// TIA Portal V16 export
// export: Created 2024-12-03T15:41:39.243873Z, ExportSetting WithDefaults, DisplayName Totally Integrated Automation Portal, DisplayVersion V16 Update 6, DisplayName TIA Portal Version Control Interface, DisplayVersion V16 Update 2, DisplayName TIA Portal Openness, DisplayVersion V16 Update 6, DisplayName TIA Portal Teamcenter Gateway, DisplayVersion V16, DisplayName SINAMICS Startdrive Advanced, DisplayVersion V16 Update 5, DisplayName SINAMICS Startdrive G130, G150, S120, S150, SINAMICS MV, S210, DisplayVersion V16 Update 5, DisplayName SINAMICS Startdrive G110M, G120, G120C, G120D, G120P, G115D, DisplayVersion V16 Update 5, DisplayName STEP 7 Professional, DisplayVersion V16 Update 6, DisplayName STEP 7 Safety, DisplayVersion V16, DisplayName WinCC Advanced / Unified PC, DisplayVersion V16 Update 6
FUNCTION_BLOCK "InputReaderConveyLinx_FB"   // FB127, SCL
{ S7_Optimized_Access := 'TRUE' }
VERSION : 0.1
// stored: AutoNumber true, IsIECCheckEnabled false, IsRetainMemResEnabled false, MemoryReserve 100, SetENOAutomatically false, UDAEnableTagReadback false
   VAR
      FTC_102_L2 : "SmartBool";
      FTC_102_L4 : "SmartBool";
      FTC_102_R2 : "SmartBool";
      FTC_102_R4 : "SmartBool";
      FTC_103_L2 : "SmartBool";
      FTC_103_L4 : "SmartBool";
      FTC_103_R2 : "SmartBool";
      FTC_103_R4 : "SmartBool";
      FTC_104_L2 : "SmartBool";
      FTC_104_L4 : "SmartBool";
      FTC_104_R2 : "SmartBool";
      FTC_104_R4 : "SmartBool";
      FTC_105_L2 : "SmartBool";
      FTC_105_L4 : "SmartBool";
      FTC_105_R2 : "SmartBool";
      FTC_105_R4 : "SmartBool";
      FTC_106_L2 : "SmartBool";
      FTC_106_L4 : "SmartBool";
      FTC_106_R2 : "SmartBool";
      FTC_106_R4 : "SmartBool";
      FTC_107_L2 : "SmartBool";
      FTC_107_L4 : "SmartBool";
      FTC_107_R2 : "SmartBool";
      FTC_107_R4 : "SmartBool";
      FTC_108_L2 : "SmartBool";
      FTC_108_L4 : "SmartBool";
      FTC_108_R2 : "SmartBool";
      FTC_108_R4 : "SmartBool";
      FTC_109_L2 : "SmartBool";
      FTC_109_L4 : "SmartBool";
      FTC_109_R2 : "SmartBool";
      FTC_109_R4 : "SmartBool";
      FTC_110_L2 : "SmartBool";
      FTC_110_L4 : "SmartBool";
      FTC_110_R2 : "SmartBool";
      FTC_110_R4 : "SmartBool";
      FTC_111_L2 : "SmartBool";
      FTC_111_L4 : "SmartBool";
      FTC_111_R2 : "SmartBool";
      FTC_111_R4 : "SmartBool";
      FTC_112_L2 : "SmartBool";
      FTC_112_L4 : "SmartBool";
      FTC_112_R2 : "SmartBool";
      FTC_112_R4 : "SmartBool";
      FTC_113_L2 : "SmartBool";
      FTC_113_L4 : "SmartBool";
      FTC_113_R2 : "SmartBool";
      FTC_113_R4 : "SmartBool";
      FTC_114_L2 : "SmartBool";
      FTC_114_L4 : "SmartBool";
      FTC_114_R2 : "SmartBool";
      FTC_114_R4 : "SmartBool";
      FTC_115_L2 : "SmartBool";
      FTC_115_L4 : "SmartBool";
      FTC_115_R2 : "SmartBool";
      FTC_115_R4 : "SmartBool";
      FTC_202_L2 : "SmartBool";
      FTC_202_L4 : "SmartBool";
      FTC_202_R2 : "SmartBool";
      FTC_202_R4 : "SmartBool";
      FTC_203_L2 : "SmartBool";
      FTC_203_L4 : "SmartBool";
      FTC_203_R2 : "SmartBool";
      FTC_203_R4 : "SmartBool";
      FTC_301_L2 : "SmartBool";
      FTC_301_L4 : "SmartBool";
      FTC_301_R2 : "SmartBool";
      FTC_301_R4 : "SmartBool";
      FTC_302_L2 : "SmartBool";
      FTC_302_L4 : "SmartBool";
      FTC_302_R2 : "SmartBool";
      FTC_302_R4 : "SmartBool";
      FTC_303_L2 : "SmartBool";
      FTC_303_L4 : "SmartBool";
      FTC_303_R2 : "SmartBool";
      FTC_303_R4 : "SmartBool";
      FTC_304_L2 : "SmartBool";
      FTC_304_L4 : "SmartBool";
      FTC_304_R2 : "SmartBool";
      FTC_304_R4 : "SmartBool";
      FTC_305_L2 : "SmartBool";
      FTC_305_L4 : "SmartBool";
      FTC_305_R2 : "SmartBool";
      FTC_305_R4 : "SmartBool";
   END_VAR
BEGIN
   REGION CON_102 

       #FTC_102_L2(I_Sensor := NOT "I_CON_102".AllSensors.LeftPin2,
                   O_data => "Inputs_DB".FTC_102_L2);

       #FTC_102_L4(I_Sensor := NOT "I_CON_102".AllSensors.LeftPin4,
                   O_data => "Inputs_DB".FTC_102_L4);

       #FTC_102_R2(I_Sensor := NOT "I_CON_102".AllSensors.RightPin2,
                   O_data => "Inputs_DB".FTC_102_R2);

       #FTC_102_R4(I_Sensor := NOT "I_CON_102".AllSensors.RightPin4,
                   O_data => "Inputs_DB".FTC_102_R4);

   END_REGION

   REGION CON_103 

       #FTC_103_L2(I_Sensor := NOT "I_CON_103".AllSensors.LeftPin2,
                   O_data => "Inputs_DB".FTC_103_L2);

       #FTC_103_L4(I_Sensor := NOT "I_CON_103".AllSensors.LeftPin4,
                   O_data => "Inputs_DB".FTC_103_L4);

       #FTC_103_R2(I_Sensor := NOT "I_CON_103".AllSensors.RightPin2,
                   O_data => "Inputs_DB".FTC_103_R2);

       #FTC_103_R4(I_Sensor := NOT "I_CON_103".AllSensors.RightPin4,
                   O_data => "Inputs_DB".FTC_103_R4);

   END_REGION

   REGION CON_104 

       #FTC_104_L2(I_Sensor := NOT "I_CON_104".AllSensors.LeftPin2,
                   O_data => "Inputs_DB".FTC_104_L2);

       #FTC_104_L4(I_Sensor := NOT "I_CON_104".AllSensors.LeftPin4,
                   O_data => "Inputs_DB".FTC_104_L4);

       #FTC_104_R2(I_Sensor := NOT "I_CON_104".AllSensors.RightPin2,
                   O_data => "Inputs_DB".FTC_104_R2);

       #FTC_104_R4(I_Sensor := NOT "I_CON_104".AllSensors.RightPin4,
                   O_data => "Inputs_DB".FTC_104_R4);

   END_REGION

   REGION CON_105 

       #FTC_105_L2(I_Sensor := NOT "I_CON_105".AllSensors.LeftPin2,
                   O_data => "Inputs_DB".FTC_105_L2);

       #FTC_105_L4(I_Sensor := NOT "I_CON_105".AllSensors.LeftPin4,
                   O_data => "Inputs_DB".FTC_105_L4);

       #FTC_105_R2(I_Sensor := NOT "I_CON_105".AllSensors.RightPin2,
                   O_data => "Inputs_DB".FTC_105_R2);

       #FTC_105_R4(I_Sensor := NOT "I_CON_105".AllSensors.RightPin4,
                   O_data => "Inputs_DB".FTC_105_R4);

   END_REGION

   REGION CON_106 

       #FTC_106_L2(I_Sensor := NOT "I_CON_106".AllSensors.LeftPin2,
                   O_data => "Inputs_DB".FTC_106_L2);

       #FTC_106_L4(I_Sensor := NOT "I_CON_106".AllSensors.LeftPin4,
                   O_data => "Inputs_DB".FTC_106_L4);

       #FTC_106_R2(I_Sensor := NOT "I_CON_106".AllSensors.RightPin2,
                   O_data => "Inputs_DB".FTC_106_R2);

       #FTC_106_R4(I_Sensor := NOT "I_CON_106".AllSensors.RightPin4,
                   O_data => "Inputs_DB".FTC_106_R4);

   END_REGION

   REGION CON_107 

       #FTC_107_L2(I_Sensor := NOT "I_CON_107".AllSensors.LeftPin2,
                   O_data => "Inputs_DB".FTC_107_L2);

       #FTC_107_L4(I_Sensor := NOT "I_CON_107".AllSensors.LeftPin4,
                   O_data => "Inputs_DB".FTC_107_L4);

       #FTC_107_R2(I_Sensor := NOT "I_CON_107".AllSensors.RightPin2,
                   O_data => "Inputs_DB".FTC_107_R2);

       #FTC_107_R4(I_Sensor := NOT "I_CON_107".AllSensors.RightPin4,
                   O_data => "Inputs_DB".FTC_107_R4);

   END_REGION

   REGION CON_108 

       #FTC_108_L2(I_Sensor := NOT "I_CON_108".AllSensors.LeftPin2,
                   O_data => "Inputs_DB".FTC_108_L2);

       #FTC_108_L4(I_Sensor := NOT "I_CON_108".AllSensors.LeftPin4,
                   O_data => "Inputs_DB".FTC_108_L4);

       #FTC_108_R2(I_Sensor := NOT "I_CON_108".AllSensors.RightPin2,
                   O_data => "Inputs_DB".FTC_108_R2);

       #FTC_108_R4(I_Sensor := NOT "I_CON_108".AllSensors.RightPin4,
                   O_data => "Inputs_DB".FTC_108_R4);

   END_REGION

   REGION CON_109 

       #FTC_109_L2(I_Sensor := NOT "I_CON_109".AllSensors.LeftPin2,
                   O_data => "Inputs_DB".FTC_109_L2);

       #FTC_109_L4(I_Sensor := NOT "I_CON_109".AllSensors.LeftPin4,
                   O_data => "Inputs_DB".FTC_109_L4);

       #FTC_109_R2(I_Sensor := NOT "I_CON_109".AllSensors.RightPin2,
                   O_data => "Inputs_DB".FTC_109_R2);

       #FTC_109_R4(I_Sensor := NOT "I_CON_109".AllSensors.RightPin4,
                   O_data => "Inputs_DB".FTC_109_R4);

   END_REGION

   REGION CON_110 

       #FTC_110_L2(I_Sensor := NOT "I_CON_110".AllSensors.LeftPin2,
                   O_data => "Inputs_DB".FTC_110_L2);

       #FTC_110_L4(I_Sensor := NOT "I_CON_110".AllSensors.LeftPin4,
                   O_data => "Inputs_DB".FTC_110_L4);

       #FTC_110_R2(I_Sensor := NOT "I_CON_110".AllSensors.RightPin2,
                   O_data => "Inputs_DB".FTC_110_R2);

       #FTC_110_R4(I_Sensor := NOT "I_CON_110".AllSensors.RightPin4,
                   O_data => "Inputs_DB".FTC_110_R4);

   END_REGION

   REGION CON_111 

       #FTC_111_L2(I_Sensor := NOT "I_CON_111".AllSensors.LeftPin2,
                   O_data => "Inputs_DB".FTC_111_L2);

       #FTC_111_L4(I_Sensor := NOT "I_CON_111".AllSensors.LeftPin4,
                   O_data => "Inputs_DB".FTC_111_L4);

       #FTC_111_R2(I_Sensor := NOT "I_CON_111".AllSensors.RightPin2,
                   O_data => "Inputs_DB".FTC_111_R2);

       #FTC_111_R4(I_Sensor := NOT "I_CON_111".AllSensors.RightPin4,
                   O_data => "Inputs_DB".FTC_111_R4);

   END_REGION

   REGION CON_112 

       #FTC_112_L2(I_Sensor := NOT "I_CON_112".AllSensors.LeftPin2,
                   O_data => "Inputs_DB".FTC_112_L2);

       #FTC_112_L4(I_Sensor := NOT "I_CON_112".AllSensors.LeftPin4,
                   O_data => "Inputs_DB".FTC_112_L4);

       #FTC_112_R2(I_Sensor := NOT "I_CON_112".AllSensors.RightPin2,
                   O_data => "Inputs_DB".FTC_112_R2);

       #FTC_112_R4(I_Sensor := NOT "I_CON_112".AllSensors.RightPin4,
                   O_data => "Inputs_DB".FTC_112_R4);

   END_REGION

   REGION CON_113 

       #FTC_113_L2(I_Sensor := NOT "I_CON_113".AllSensors.LeftPin2,
                   O_data => "Inputs_DB".FTC_113_L2);

       #FTC_113_L4(I_Sensor := NOT "I_CON_113".AllSensors.LeftPin4,
                   O_data => "Inputs_DB".FTC_113_L4);

       #FTC_113_R2(I_Sensor := NOT "I_CON_113".AllSensors.RightPin2,
                   O_data => "Inputs_DB".FTC_113_R2);

       #FTC_113_R4(I_Sensor := NOT "I_CON_113".AllSensors.RightPin4,
                   O_data => "Inputs_DB".FTC_113_R4);

   END_REGION

   REGION CON_114 

       #FTC_114_L2(I_Sensor := NOT "I_CON_114".AllSensors.LeftPin2,
                   O_data => "Inputs_DB".FTC_114_L2);

       #FTC_114_L4(I_Sensor := NOT "I_CON_114".AllSensors.LeftPin4,
                   O_data => "Inputs_DB".FTC_114_L4);

       #FTC_114_R2(I_Sensor := NOT "I_CON_114".AllSensors.RightPin2,
                   O_data => "Inputs_DB".FTC_114_R2);

       #FTC_114_R4(I_Sensor := NOT "I_CON_114".AllSensors.RightPin4,
                   O_data => "Inputs_DB".FTC_114_R4);

   END_REGION

   REGION CON_115 

       #FTC_115_L2(I_Sensor := NOT "I_CON_115".AllSensors.LeftPin2,
                   O_data => "Inputs_DB".FTC_115_L2);

       #FTC_115_L4(I_Sensor := NOT "I_CON_115".AllSensors.LeftPin4,
                   O_data => "Inputs_DB".FTC_115_L4);

       #FTC_115_R2(I_Sensor := NOT "I_CON_115".AllSensors.RightPin2,
                   O_data => "Inputs_DB".FTC_115_R2);

       #FTC_115_R4(I_Sensor := NOT "I_CON_115".AllSensors.RightPin4,
                   O_data => "Inputs_DB".FTC_115_R4);

   END_REGION

   REGION CON_202 

       #FTC_202_L2(I_Sensor := NOT "I_CON_202".AllSensors.LeftPin2,
                   O_data => "Inputs_DB".FTC_202_L2);

       #FTC_202_L4(I_Sensor := NOT "I_CON_202".AllSensors.LeftPin4,
                   O_data => "Inputs_DB".FTC_202_L4);

       #FTC_202_R2(I_Sensor := NOT "I_CON_202".AllSensors.RightPin2,
                   O_data => "Inputs_DB".FTC_202_R2);

       #FTC_202_R4(I_Sensor := NOT "I_CON_202".AllSensors.RightPin4,
                   O_data => "Inputs_DB".FTC_202_R4);

   END_REGION

   REGION CON_203 

       #FTC_203_L2(I_Sensor := NOT "I_CON_203".AllSensors.LeftPin2,
                   O_data => "Inputs_DB".FTC_203_L2);

       #FTC_203_L4(I_Sensor := NOT "I_CON_203".AllSensors.LeftPin4,
                   O_data => "Inputs_DB".FTC_203_L4);

       #FTC_203_R2(I_Sensor := NOT "I_CON_203".AllSensors.RightPin2,
                   O_data => "Inputs_DB".FTC_203_R2);

       #FTC_203_R4(I_Sensor := NOT "I_CON_203".AllSensors.RightPin4,
                   O_data => "Inputs_DB".FTC_203_R4);

   END_REGION

   REGION CON_301 

       #FTC_301_L2(I_Sensor := NOT "I_CON_301".AllSensors.LeftPin2,
                   O_data => "Inputs_DB".FTC_301_L2);

       #FTC_301_L4(I_Sensor := NOT "I_CON_301".AllSensors.LeftPin4,
                   O_data => "Inputs_DB".FTC_301_L4);

       #FTC_301_R2(I_Sensor := NOT "I_CON_301".AllSensors.RightPin2,
                   O_data => "Inputs_DB".FTC_301_R2);

       #FTC_301_R4(I_Sensor := NOT "I_CON_301".AllSensors.RightPin4,
                   O_data => "Inputs_DB".FTC_301_R4);

   END_REGION

   REGION CON_302 

       #FTC_302_L2(I_Sensor := NOT "I_CON_302".AllSensors.LeftPin2,
                   O_data => "Inputs_DB".FTC_302_L2);

       #FTC_302_L4(I_Sensor := NOT "I_CON_302".AllSensors.LeftPin4,
                   O_data => "Inputs_DB".FTC_302_L4);

       #FTC_302_R2(I_Sensor := NOT "I_CON_302".AllSensors.RightPin2,
                   O_data => "Inputs_DB".FTC_302_R2);

       #FTC_302_R4(I_Sensor := NOT "I_CON_302".AllSensors.RightPin4,
                   O_data => "Inputs_DB".FTC_302_R4);

   END_REGION

   REGION CON_303 

       #FTC_303_L2(I_Sensor := NOT "I_CON_303".AllSensors.LeftPin2,
                   O_data => "Inputs_DB".FTC_303_L2);

       #FTC_303_L4(I_Sensor := NOT "I_CON_303".AllSensors.LeftPin4,
                   O_data => "Inputs_DB".FTC_303_L4);

       #FTC_303_R2(I_Sensor := NOT "I_CON_303".AllSensors.RightPin2,
                   O_data => "Inputs_DB".FTC_303_R2);

       #FTC_303_R4(I_Sensor := NOT "I_CON_303".AllSensors.RightPin4,
                   O_data => "Inputs_DB".FTC_303_R4);

   END_REGION

   REGION CON_304 

       #FTC_304_L2(I_Sensor := NOT "I_CON_304".AllSensors.LeftPin2,
                   O_data => "Inputs_DB".FTC_304_L2);

       #FTC_304_L4(I_Sensor := NOT "I_CON_304".AllSensors.LeftPin4,
                   O_data => "Inputs_DB".FTC_304_L4);

       #FTC_304_R2(I_Sensor := NOT "I_CON_304".AllSensors.RightPin2,
                   O_data => "Inputs_DB".FTC_304_R2);

       #FTC_304_R4(I_Sensor := NOT "I_CON_304".AllSensors.RightPin4,
                   O_data => "Inputs_DB".FTC_304_R4);

   END_REGION

   REGION CON_305 

       #FTC_305_L2(I_Sensor := NOT "I_CON_305".AllSensors.LeftPin2,
                   O_data => "Inputs_DB".FTC_305_L2);

       #FTC_305_L4(I_Sensor := NOT "I_CON_305".AllSensors.LeftPin4,
                   O_data => "Inputs_DB".FTC_305_L4);

       #FTC_305_R2(I_Sensor := NOT "I_CON_305".AllSensors.RightPin2,
                   O_data => "Inputs_DB".FTC_305_R2);

       #FTC_305_R4(I_Sensor := NOT "I_CON_305".AllSensors.RightPin4,
                   O_data => "Inputs_DB".FTC_305_R4);

   END_REGION
END_FUNCTION_BLOCK
